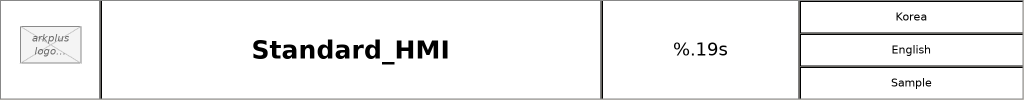
VISUALIZATION UpperBar  // 1024x100
    Rectangle (0,0 100x99)
    Image (20,26 61x37), image: arkplus logo_Resize
    Rectangle (101,0 500x99), "Standard_HMI"
    Rectangle (602,0 197x99), "%.19s", text variable: GVL_HMI.sCurrentTime
    Rectangle (800,1 223x32), "Korea"
        OnMouseClick: ChangeLanguage ChangeLanguage=Korea
    Rectangle (800,34 223x32), "English"
        OnMouseClick: ChangeLanguage ChangeLanguage=English
    Rectangle (800,67 223x32), "Sample"
END_VISUALIZATION

(* stored: Version 1.1.0.1
   Visu UpperBar: Id {522e1359-ba2b-4c1d-a40e-8279e71f4ccb} *)
